FUNCTION_BLOCK FB_LamparaTemporizada_SFC
VAR_INPUT
    TiempoEncendido: REAL := 2.0;
END_VAR
VAR_OUTPUT
    TiempoPendiente: REAL;
END_VAR
VAR
    Lampara AT %Q*: BOOL;
    Pulsador AT %I*: BOOL;
END_VAR

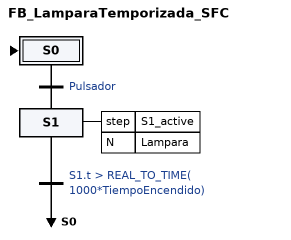
INITIAL_STEP S0:
END_STEP
TRANSITION FROM S0 TO S1
    := Pulsador;
END_TRANSITION
STEP S1:
    S1_active(N);  // step action
    Lampara(N);
END_STEP
TRANSITION FROM S1 TO S0
    := S1.t > REAL_TO_TIME(1000*TiempoEncendido);
END_TRANSITION

ACTION S1_active:
TiempoPendiente := TiempoEncendido - (TIME_TO_REAL(S1.t)/1000);
END_ACTION

END_FUNCTION_BLOCK

(* stored: Version 1.1.0.1, ProductVersion 3.1.4024.15
   POU FB_LamparaTemporizada_SFC: Id {9fc26670-06c3-48c6-bf53-687a17a3ed03}, SpecialFunc None
   Action S1_active: Id {6203564d-ab62-43c5-974f-a3b810bc5fc3} *)
